Staubli VAL3: findLastPathPos.pgx

program findLastPathPos(string x_sPath (dimensions=1), num& x_nPos[] (dimensions=1))
  local num l_nPos[2]
  local string l_sPath
begin
  // get the trajType
  l_sPath=x_sPath
  x_nPos=0
  do
    l_nPos=find(l_sPath,"/")
    if l_nPos==-1
      l_nPos=find(l_sPath,"\")
    endIf
    if l_nPos!=-1
      x_nPos=x_nPos+l_nPos+1
      l_nPos[1]=l_nPos
      l_sPath=right(l_sPath,len(l_sPath)-l_nPos-1)
    endIf
  until l_nPos==-1
  // came back one
  x_nPos=x_nPos-l_nPos[1]-1
end
